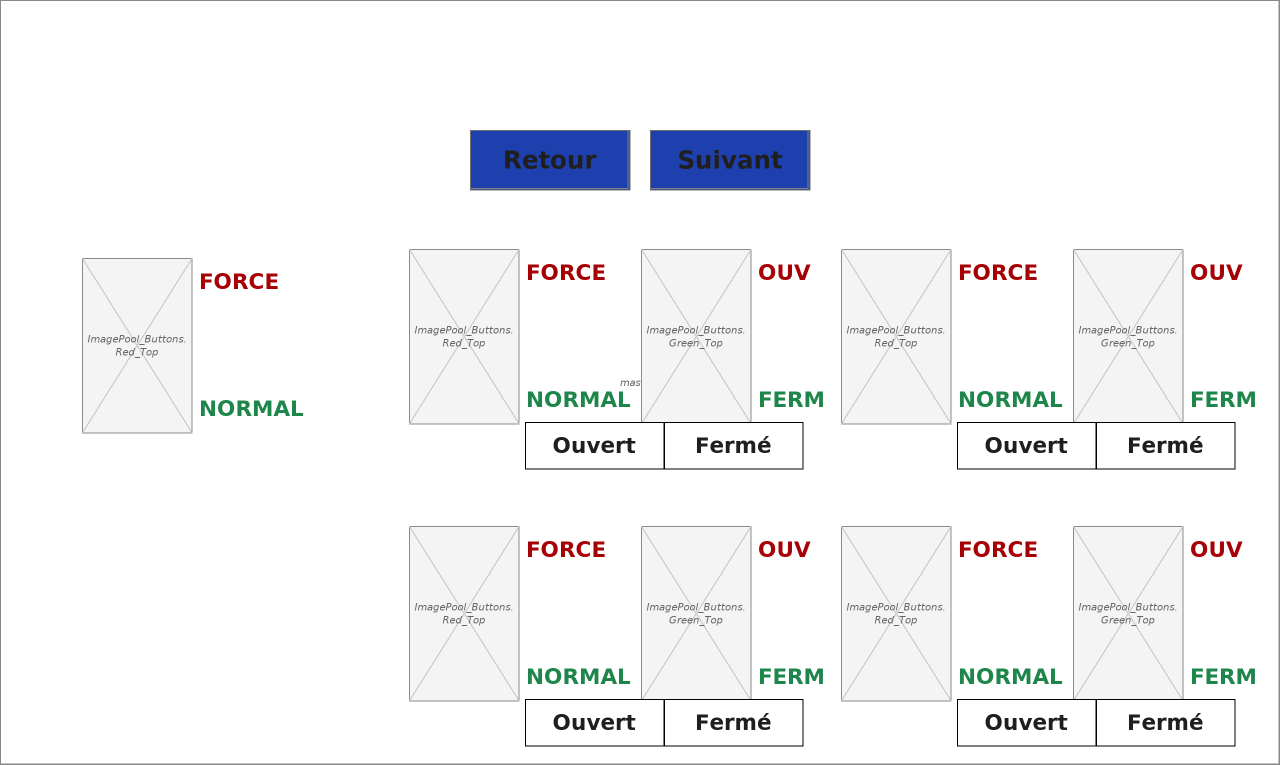
VISUALIZATION Maintenance_3  // 1280x765
    Frame (0,0 1280x765)
        shows masque()
    Group (409,209 415x260), invisible if: NOT Option_Bas_Debit
        Group (0,40 415x173)
            Group (0,0 232x174)
                Group (0,0 110x175)
                    Image (0,0 110x175), invisible if: EF_Vanne_Souf_Bas_Deb, image: ImagePool_Buttons.Green_Bottom
                        OnMouseDown: toggle EF_Vanne_Souf_Bas_Deb
                    Image (0,0 110x175), invisible if: NOT EF_Vanne_Souf_Bas_Deb, image: ImagePool_Buttons.Red_Top
                        OnMouseDown: toggle EF_Vanne_Souf_Bas_Deb
                Rectangle (114,0 118x47), "FORCE"
                Rectangle (114,63 118x47), "MODE"
                Rectangle (114,127 118x47), "NORMAL"
            Group (232,0 196x174), invisible if: NOT EF_Vanne_Souf_Bas_Deb
                Group (0,0 110x175)
                    Image (0,0 110x175), invisible if: F_Vanne_Souf_Bas_Deb, image: ImagePool_Buttons.Red_Bottom
                        OnMouseDown: toggle F_Vanne_Souf_Bas_Deb
                    Image (0,0 110x175), invisible if: NOT F_Vanne_Souf_Bas_Deb, image: ImagePool_Buttons.Green_Top
                        OnMouseDown: toggle F_Vanne_Souf_Bas_Deb
                Rectangle (114,0 82x47), "OUV"
                Rectangle (114,63 82x47), "OUT"
                Rectangle (114,127 82x47), "FERM"
        Group (33,213 350x47)
            Rectangle (0,0 83x47), "FDC :"
            RoundedRectangle (83,0 139x47), "Ouvert", invisible if: NOT E_Vanne_Souf_Bas_Deb_Ouv
            RoundedRectangle (222,0 139x47), "Fermé", invisible if: NOT E_Vanne_Souf_Bas_Deb_Ferm
        Rectangle (0,0 415x40), "Soufflage bas débit"
    Group (409,486 415x260), invisible if: NOT Option_Bas_Debit
        Group (0,40 415x173)
            Group (0,0 232x174)
                Group (0,0 110x175)
                    Image (0,0 110x175), invisible if: EF_Vanne_Ext_Bas_Deb, image: ImagePool_Buttons.Green_Bottom
                        OnMouseDown: toggle EF_Vanne_Ext_Bas_Deb
                    Image (0,0 110x175), invisible if: NOT EF_Vanne_Ext_Bas_Deb, image: ImagePool_Buttons.Red_Top
                        OnMouseDown: toggle EF_Vanne_Ext_Bas_Deb
                Rectangle (114,0 118x47), "FORCE"
                Rectangle (114,63 118x47), "MODE"
                Rectangle (114,127 118x47), "NORMAL"
            Group (232,0 196x174), text variable: NOT EF_Vanne_Ext_Bas_Deb, invisible if: NOT EF_Vanne_Ext_Bas_Deb
                Group (0,0 110x175)
                    Image (0,0 110x175), invisible if: F_Vanne_Ext_Bas_Deb, image: ImagePool_Buttons.Red_Bottom
                        OnMouseDown: toggle F_Vanne_Ext_Bas_Deb
                    Image (0,0 110x175), invisible if: NOT F_Vanne_Ext_Bas_Deb, image: ImagePool_Buttons.Green_Top
                        OnMouseDown: toggle F_Vanne_Ext_Bas_Deb
                Rectangle (114,0 82x47), "OUV"
                Rectangle (114,63 82x47), "OUT"
                Rectangle (114,127 82x47), "FERM"
        Group (33,213 350x47)
            Rectangle (0,0 83x47), "FDC :"
            RoundedRectangle (83,0 139x47), "Ouvert", invisible if: NOT E_Vanne_Ext_Bas_Deb_Ouv
            RoundedRectangle (222,0 139x47), "Fermé", invisible if: NOT E_Vanne_Ext_Bas_Deb_Ferm
        Rectangle (0,0 415x40), "Extraction bas débit"
    Group (841,209 415x260), invisible if: NOT Option_Douchette
        Group (0,40 415x173)
            Group (0,0 232x174)
                Group (0,0 110x175)
                    Image (0,0 110x175), invisible if: EF_Cmd_Vanne_Alim_Douchette, image: ImagePool_Buttons.Green_Bottom
                        OnMouseDown: toggle EF_Cmd_Vanne_Alim_Douchette
                    Image (0,0 110x175), invisible if: NOT EF_Cmd_Vanne_Alim_Douchette, image: ImagePool_Buttons.Red_Top
                        OnMouseDown: toggle EF_Cmd_Vanne_Alim_Douchette
                Rectangle (114,0 118x47), "FORCE"
                Rectangle (114,63 118x47), "MODE"
                Rectangle (114,127 118x47), "NORMAL"
            Group (232,0 196x174), invisible if: NOT EF_Cmd_Vanne_Alim_Douchette
                Group (0,0 110x175)
                    Image (0,0 110x175), invisible if: F_Cmd_Vanne_Alim_Douchette, image: ImagePool_Buttons.Red_Bottom
                        OnMouseDown: toggle F_Cmd_Vanne_Alim_Douchette
                    Image (0,0 110x175), invisible if: NOT F_Cmd_Vanne_Alim_Douchette, image: ImagePool_Buttons.Green_Top
                        OnMouseDown: toggle F_Cmd_Vanne_Alim_Douchette
                Rectangle (114,0 82x47), "OUV"
                Rectangle (114,63 82x47), "OUT"
                Rectangle (114,127 82x47), "FERM"
        Group (33,213 350x47)
            Rectangle (0,0 83x47), "FDC :"
            RoundedRectangle (83,0 139x47), "Ouvert", invisible if: NOT E_Vanne_Alim_Douchette_Ouv
            RoundedRectangle (222,0 139x47), "Fermé", invisible if: NOT E_Vanne_Alim_Douchette_Ferm
        Rectangle (0,0 415x40), "Douchette"
    Group (841,486 415x260), invisible if: NOT Option_NEP
        Group (0,40 415x173)
            Group (0,0 232x174)
                Group (0,0 110x175)
                    Image (0,0 110x175), invisible if: EF_Vanne_Alim_NEP, image: ImagePool_Buttons.Green_Bottom
                        OnMouseDown: toggle EF_Vanne_Alim_NEP
                    Image (0,0 110x175), invisible if: NOT EF_Vanne_Alim_NEP, image: ImagePool_Buttons.Red_Top
                        OnMouseDown: toggle EF_Vanne_Alim_NEP
                Rectangle (114,0 118x47), "FORCE"
                Rectangle (114,63 118x47), "MODE"
                Rectangle (114,127 118x47), "NORMAL"
            Group (232,0 196x174), invisible if: NOT EF_Vanne_Alim_NEP
                Group (0,0 110x175)
                    Image (0,0 110x175), invisible if: F_Vanne_Alim_NEP, image: ImagePool_Buttons.Red_Bottom
                        OnMouseDown: toggle F_Vanne_Alim_NEP
                    Image (0,0 110x175), invisible if: NOT F_Vanne_Alim_NEP, image: ImagePool_Buttons.Green_Top
                        OnMouseDown: toggle F_Vanne_Alim_NEP
                Rectangle (114,0 82x47), "OUV"
                Rectangle (114,63 82x47), "OUT"
                Rectangle (114,127 82x47), "FERM"
        Group (33,213 350x47)
            Rectangle (0,0 83x47), "FDC :"
            RoundedRectangle (83,0 139x47), "Ouvert", invisible if: NOT E_Vanne_Alim_NEP_Ouv
            RoundedRectangle (222,0 139x47), "Fermé", invisible if: NOT E_Vanne_Alim_NEP_Ferm
        Rectangle (0,0 415x40), "Vanne NEP"
    Button (650,130 160x60), "Suivant"
        OnMouseDown: execute {
            IF (Option_WC_GV OR Option_WC_PV OR Option_Prise)
            	THEN
            	VisuElems.CURRENTVISU := 'Maintenance_4';
            	ELSIF (Option_Cabine_Climatique)
            		THEN
            		VisuElems.CURRENTVISU := 'Maintenance_5';
            	ELSIF (Option_Com_RegSouf_Ultrason)
            		THEN
            		VisuElems.CURRENTVISU := 'Maintenance_6';
            	ELSE
            		VisuElems.CURRENTVISU := 'Maintenance_7';
            END_IF
        }
    Button (470,130 160x60), "Retour"
        OnMouseDown: execute {
            IF (Option_Douche OR Option_Lavabo)
            	THEN
            	VisuElems.CURRENTVISU := 'Maintenance_2';
            	ELSIF (Option_RegSouf_Ultrason OR Option_Reg_Etanche_Ext OR Option_V3V_EauMitig)
            		THEN
            		VisuElems.CURRENTVISU := 'Maintenance_1';
            	ELSE
            	VisuElems.CURRENTVISU := 'menu';
            END_IF
        }
    Group (15,204 380x545), invisible if: NOT Option_Bas_Debit
        Rectangle (0,0 379x63), "Moteur bas débit"
        Group (67,54 245x174)
            Group (0,0 110x175)
                Image (0,0 110x175), invisible if: Tab_Mot_Aerobox_Bas_Deb.Mot_Ecriture.0, image: ImagePool_Buttons.Green_Bottom
                    OnMouseDown: toggle Tab_Mot_Aerobox_Bas_Deb.Mot_Ecriture.0
                Image (0,0 110x175), invisible if: NOT Tab_Mot_Aerobox_Bas_Deb.Mot_Ecriture.0, image: ImagePool_Buttons.Red_Top
                    OnMouseDown: toggle Tab_Mot_Aerobox_Bas_Deb.Mot_Ecriture.0
            Rectangle (114,0 131x47), "FORCE"
            Rectangle (111,63 131x47), "MODE"
            Rectangle (114,127 131x47), "NORMAL"
        Rectangle (26,292 327x63), "Appli : %.0f %%", text variable: Cons_Actionneur_Moteur_BasDebit
        Rectangle (26,355 327x63), "Mesure : %.0f m3/h", text variable: MES_Petit_Debit_m3h_Extraction
        RoundedRectangle (2,228 374x63), "Vitesse : %.0f %%", text variable: Tab_Mot_Aerobox_Bas_Deb.W_ConsForcage, invisible if: NOT Tab_Mot_Aerobox_Bas_Deb.Mot_Ecriture.0
            OnMouseDown: write the text variable via VisuDialogs.Numpad, min 0, max 100, format %.0f
        RoundedRectangle (2,418 374x63), "Vit Max : %.0f %%", text variable: Tab_Mot_Aerobox_Bas_Deb.W_LimiteMaxCons
            OnMouseDown: write the text variable via VisuDialogs.Numpad, min 0, max 100, format %.0f
        RoundedRectangle (2,482 374x63), "Vit Min : %.0f %%", text variable: Tab_Mot_Aerobox_Bas_Deb.W_LimiteMinCons
            OnMouseDown: write the text variable via VisuDialogs.Numpad, min 0, max 100, format %.0f
END_VISUALIZATION

(* stored: Version 1.1.0.1, ProductVersion 3.1.4024.15
   Visu Maintenance_3: Id {1fac4cb1-5616-4523-9c19-c251714eafd3} *)
